TYPE ST_CalibrationReportListItem :
STRUCT
	sReportId       : STRING(50);
    sCalibrationNo  : STRING(30);
    sCreatedAt      : STRING(30);
    sUserId         : STRING(50);
END_STRUCT
END_TYPE

(* stored: Version 1.1.0.1, ProductVersion 3.1.4024.15
   DUT ST_CalibrationReportListItem: Id {e2253b3d-bdb0-4a19-b4d2-9e01d5c49bee} *)
